// TIA Portal project "定时器练习，控制主轴电机和油泵电机的1顺序启停_V16" (V16)

(* hardware
DEVICE "S7-1200 station_1"  S7-1200 Station
   slot 0: "Rack_0"  S7-1200 Rack  Rack  V1.0
   slot 1: "PLC_1"  CPU 1214C DC/DC/DC  6ES7 214-1AG40-0XB0  V4.2
DEVICE "HMI_1"  KTP700 Basic PN
   slot 0: "HMI_1"  KTP700 Basic PN  6AV2 123-2GB03-0AX0  15.1.0.0
   slot 1: "HMI_RT_1"  KTP700 Basic PN  6AV2 123-2GB03-0AX0  15.1.0.0
   slot 5: "HMI_1.IE_CP_1"  PROFINET Interface  15.0.1.0
      slot 1: "PROFINET Interface_1"  PROFINET Interface
         slot 1: "Port_1"  Port
*)

// ===== PLC "PLC_1"  CPU 1214C DC/DC/DC =====

VAR_GLOBAL   // PLC tag table "默认变量表"
   "启动上升沿信号" AT %M0.0 : Bool;
   "油泵启动标志" AT %M0.1 : Bool;
   "启动电机延时信号" AT %MD200 : Time;
   "主轴标志" AT %M0.2 : Bool;
   "急停下降沿信号" AT %M0.3 : Bool;
   "油泵停止标志" AT %M0.4 : Bool;
   "主轴停止延时" AT %MD2004 : Time;
   "油泵停止标志(1)" AT %M0.5 : Bool;
   "上一个扫描周期" AT %M10.0 : Bool;
   "主轴标志1" AT %M10.1 : Bool;
   "油泵停止扫描周期" AT %M0.6 : Bool;
   "Tag_1" AT %M20.0 : Bool;
   "Tag_2" AT %M20.1 : Bool;
   "Tag_3" AT %M20.2 : Bool;
   "Tag_4" AT %M30.0 : Bool;
   "Tag_5" AT %M30.1 : Bool;
   "Tag_6" AT %M20.4 : Bool;
   "Tag_7" AT %M20.3 : Bool;
   "系统运行指示灯标志1" AT %M40.0 : Bool;
   "系统运行指示灯标志2" AT %M40.1 : Bool;
   "Tag_8" AT %MD300 : Time;
   "Tag_9" AT %MD304 : Time;
   "Tag_10" AT %MD308 : Time;
   "Tag_11" AT %MD312 : Time;
   "系统停止运行标志1" AT %M40.2 : Bool;
END_VAR

VAR_GLOBAL   // PLC tag table "io表"
   "启动" AT %I0.0 : Bool;
   "停止" AT %I0.1 : Bool;
   "正转" AT %I0.2 : Bool;
   "反转" AT %I0.3 : Bool;
   "急停" AT %I0.4 : Bool;
   "主轴急停" AT %I0.5 : Bool;
   "油泵电机急停" AT %I0.6 : Bool;
   "主轴继电器" AT %Q0.0 : Bool;
   "油泵继电器" AT %Q0.1 : Bool;
   "主轴正转" AT %Q0.2 : Bool;
   "主轴反转" AT %Q0.3 : Bool;
   "系统运行指示灯" AT %Q0.4 : Bool;
   "系统停止指示灯" AT %Q0.5 : Bool;
   "主轴运行指示灯" AT %Q0.6 : Bool;
   "油泵运行指示灯" AT %Q0.7 : Bool;
END_VAR

VAR_GLOBAL   // PLC tag table "触摸屏变量"
   "触摸屏启动" AT %M100.0 : Bool;
   "触摸屏停止" AT %M100.1 : Bool;
   "触摸屏急停" AT %M100.2 : Bool;
   "触摸屏正转" AT %M100.3 : Bool;
   "触摸屏反转" AT %M100.4 : Bool;
   "触摸屏正转急停" AT %M100.5 : Bool;
   "触摸屏反转急停" AT %M100.6 : Bool;
END_VAR

// folder: System blocks/Program resources

DATA_BLOCK "IEC_Timer_0_DB"   // DB1
{ S7_Optimized_Access := 'TRUE' }
AUTHOR : Simatic
FAMILY : IEC
NAME : IEC_TMR
VERSION : 1.0
// stored: InstanceOfName IEC_TIMER
"IEC_TIMER"
BEGIN
END_DATA_BLOCK

DATA_BLOCK "IEC_Timer_0_DB_1"   // DB2
{ S7_Optimized_Access := 'TRUE' }
AUTHOR : Simatic
FAMILY : IEC
NAME : IEC_TMR
VERSION : 1.0
// stored: InstanceOfName IEC_TIMER
"IEC_TIMER"
BEGIN
END_DATA_BLOCK

DATA_BLOCK "IEC_Timer_0_DB_2"   // DB3
{ S7_Optimized_Access := 'TRUE' }
AUTHOR : Simatic
FAMILY : IEC
NAME : IEC_TMR
VERSION : 1.0
// stored: InstanceOfName IEC_TIMER
"IEC_TIMER"
BEGIN
END_DATA_BLOCK

DATA_BLOCK "IEC_Timer_0_DB_3"   // DB4
{ S7_Optimized_Access := 'TRUE' }
AUTHOR : Simatic
FAMILY : IEC
NAME : IEC_TMR
VERSION : 1.0
// stored: InstanceOfName IEC_TIMER
"IEC_TIMER"
BEGIN
END_DATA_BLOCK

DATA_BLOCK "IEC_Timer_0_DB_4"   // DB5
{ S7_Optimized_Access := 'TRUE' }
AUTHOR : Simatic
FAMILY : IEC
NAME : IEC_TMR
VERSION : 1.0
// stored: InstanceOfName IEC_TIMER
"IEC_TIMER"
BEGIN
END_DATA_BLOCK

DATA_BLOCK "IEC_Timer_0_DB_5"   // DB6
{ S7_Optimized_Access := 'TRUE' }
AUTHOR : Simatic
FAMILY : IEC
NAME : IEC_TMR
VERSION : 1.0
// stored: InstanceOfName IEC_TIMER
"IEC_TIMER"
BEGIN
END_DATA_BLOCK

// folder: (top level)

ORGANIZATION_BLOCK "Main"   // OB1, LAD, ProgramCycle
TITLE = "Main Program Sweep (Cycle)"
{ S7_Optimized_Access := 'TRUE' }
VERSION : 0.1
   VAR_INPUT
      Initial_Call : Bool;   // Initial call of this OB
      Remanence : Bool;   // =True, if remanent data are available
   END_VAR
   VAR_TEMP   // added for the SCL form of the ladder/FBD networks
      _w1 : Bool;
      _w2 : Bool;
      _w3 : Bool;
      _w4 : Bool;
   END_VAR
BEGIN

REGION Network 1: 启动系统
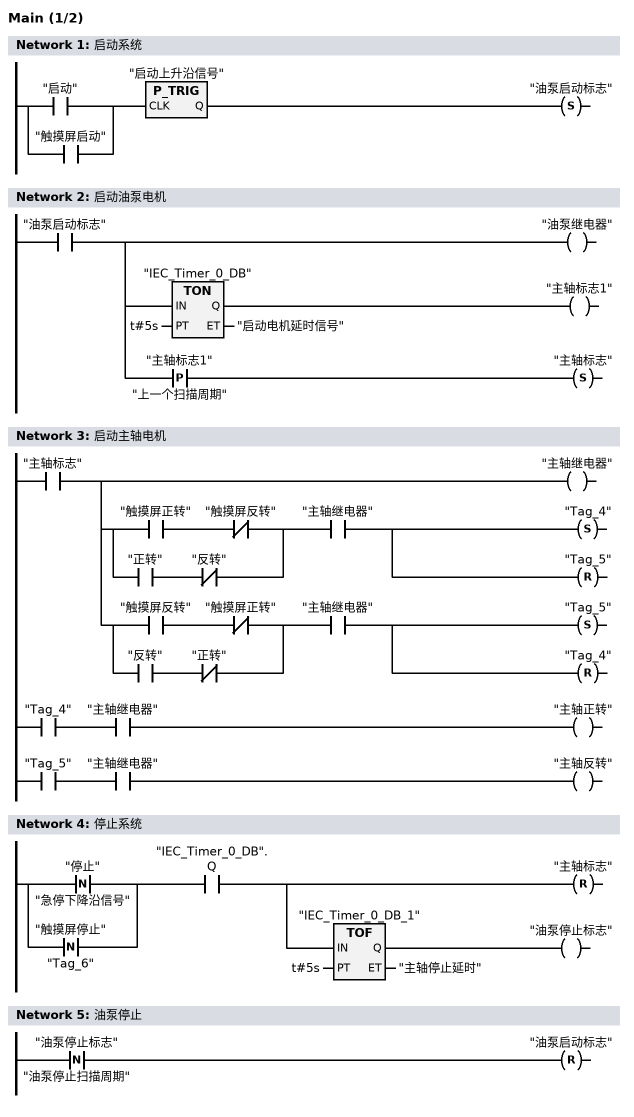
   RUNG wire#powerrail
      Contact( "启动" )
      wire#w1
      P_Trig( "启动上升沿信号" )
      S_Coil( "油泵启动标志" )
   END_RUNG
   RUNG wire#powerrail
      Contact( "触摸屏启动" )
   END_RUNG wire#w1
   // the same network as SCL:
   #_w1 := "启动" OR "触摸屏启动";
   #_w2 := #_w1 AND NOT "启动上升沿信号";   // rising edge
   "启动上升沿信号" := #_w1;
   IF #_w2 THEN "油泵启动标志" := TRUE; END_IF;
END_REGION

REGION Network 2: 启动油泵电机
   "油泵继电器" := "油泵启动标志";
   "IEC_Timer_0_DB".TON(IN := "油泵启动标志", PT := t#5s, ET => "启动电机延时信号");
   "主轴标志1" := "IEC_Timer_0_DB".Q;
   #_w1 := "油泵启动标志" AND "主轴标志1" AND NOT "上一个扫描周期";   // rising edge of "主轴标志1"
   "上一个扫描周期" := "主轴标志1";
   IF #_w1 THEN "主轴标志" := TRUE; END_IF;
END_REGION

REGION Network 3: 启动主轴电机
   RUNG wire#powerrail
      Contact( "主轴标志" )
      wire#w1
      Coil( "主轴继电器" )
   END_RUNG
   RUNG wire#w1
      Contact( "触摸屏正转" )
      I_Contact( "触摸屏反转" )
      wire#w2
      Contact( "主轴继电器" )
      wire#w3
      S_Coil( "Tag_4" )
   END_RUNG
   RUNG wire#w1
      Contact( "正转" )
      I_Contact( "反转" )
   END_RUNG wire#w2
   RUNG wire#w3
      R_Coil( "Tag_5" )
   END_RUNG
   RUNG wire#w1
      Contact( "触摸屏反转" )
      I_Contact( "触摸屏正转" )
      wire#w4
      Contact( "主轴继电器" )
      wire#w5
      S_Coil( "Tag_5" )
   END_RUNG
   RUNG wire#w1
      Contact( "反转" )
      I_Contact( "正转" )
   END_RUNG wire#w4
   RUNG wire#w5
      R_Coil( "Tag_4" )
   END_RUNG
   RUNG wire#powerrail
      Contact( "Tag_4" )
      Contact( "主轴继电器" )
      Coil( "主轴正转" )
   END_RUNG
   RUNG wire#powerrail
      Contact( "Tag_5" )
      Contact( "主轴继电器" )
      Coil( "主轴反转" )
   END_RUNG
   // the same network as SCL:
   "主轴继电器" := "主轴标志";
   IF "主轴标志" AND (("触摸屏正转" AND NOT "触摸屏反转") OR ("正转" AND NOT "反转")) AND "主轴继电器" THEN
       "Tag_4" := TRUE;
       "Tag_5" := FALSE;
   END_IF;
   IF "主轴标志" AND (("触摸屏反转" AND NOT "触摸屏正转") OR ("反转" AND NOT "正转")) AND "主轴继电器" THEN
       "Tag_5" := TRUE;
       "Tag_4" := FALSE;
   END_IF;
   "主轴正转" := "Tag_4" AND "主轴继电器";
   "主轴反转" := "Tag_5" AND "主轴继电器";
END_REGION

REGION Network 4: 停止系统
   #_w1 := NOT "停止" AND "急停下降沿信号";   // falling edge of "停止"
   "急停下降沿信号" := "停止";
   #_w2 := NOT "触摸屏停止" AND "Tag_6";   // falling edge of "触摸屏停止"
   "Tag_6" := "触摸屏停止";
   #_w3 := (#_w1 OR #_w2) AND "IEC_Timer_0_DB".Q;
   IF #_w3 THEN "主轴标志" := FALSE; END_IF;
   "IEC_Timer_0_DB_1".TOF(IN := #_w3, PT := t#5s, ET => "主轴停止延时");
   "油泵停止标志" := "IEC_Timer_0_DB_1".Q;
END_REGION

REGION Network 5: 油泵停止
   RUNG wire#powerrail
      N_Contact(operand := "油泵停止标志", bit := "油泵停止扫描周期")
      R_Coil( "油泵启动标志" )
   END_RUNG
   // the same network as SCL:
   #_w1 := NOT "油泵停止标志" AND "油泵停止扫描周期";   // falling edge of "油泵停止标志"
   "油泵停止扫描周期" := "油泵停止标志";
   IF #_w1 THEN "油泵启动标志" := FALSE; END_IF;
END_REGION

REGION Network 6: 急停
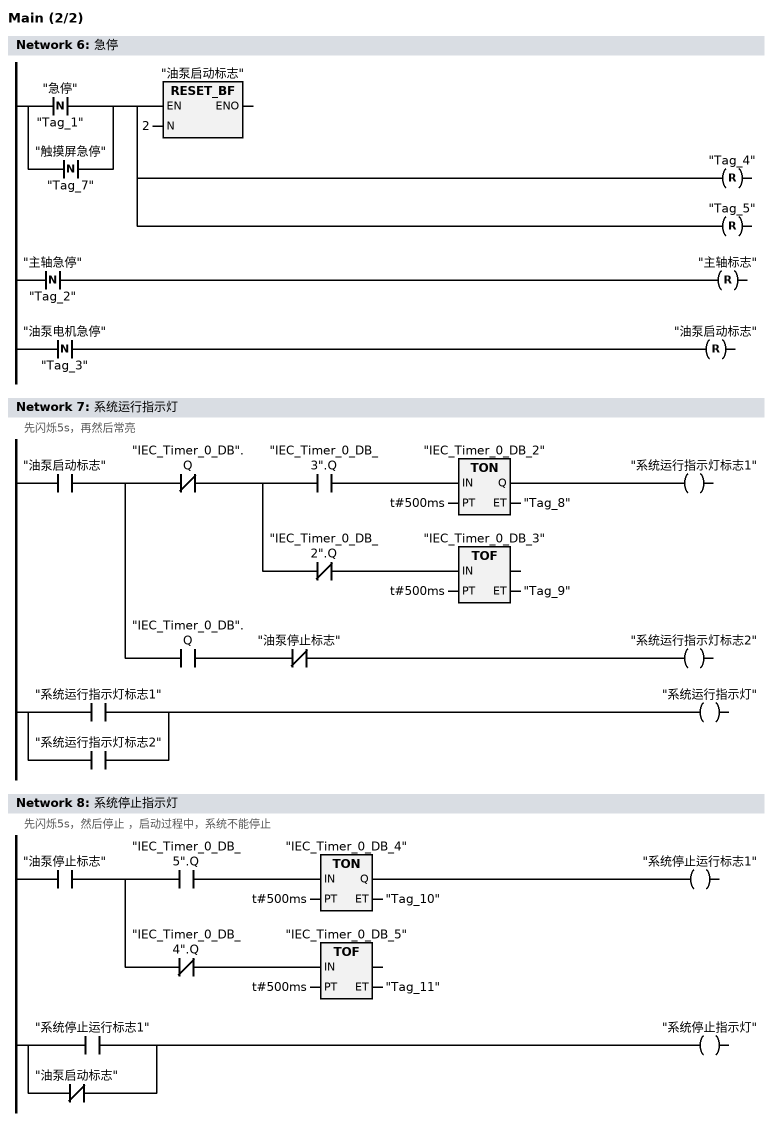
   // no SCL statement known for RBitfield: written as a call
   #_w1 := NOT "急停" AND "Tag_1";   // falling edge of "急停"
   "Tag_1" := "急停";
   #_w2 := NOT "触摸屏急停" AND "Tag_7";   // falling edge of "触摸屏急停"
   "Tag_7" := "触摸屏急停";
   IF #_w1 OR #_w2 THEN
       RESET_BF(operand := "油泵启动标志", n := 2);
       "Tag_4" := FALSE;
       "Tag_5" := FALSE;
   END_IF;
   #_w3 := NOT "主轴急停" AND "Tag_2";   // falling edge of "主轴急停"
   "Tag_2" := "主轴急停";
   IF #_w3 THEN "主轴标志" := FALSE; END_IF;
   #_w4 := NOT "油泵电机急停" AND "Tag_3";   // falling edge of "油泵电机急停"
   "Tag_3" := "油泵电机急停";
   IF #_w4 THEN "油泵启动标志" := FALSE; END_IF;
END_REGION

REGION Network 7: 系统运行指示灯
   // 先闪烁5s，再然后常亮
   #_w1 := "油泵启动标志" AND NOT "IEC_Timer_0_DB".Q;
   "IEC_Timer_0_DB_2".TON(IN := #_w1 AND "IEC_Timer_0_DB_3".Q, PT := t#500ms, ET => "Tag_8");
   "系统运行指示灯标志1" := "IEC_Timer_0_DB_2".Q;
   "IEC_Timer_0_DB_3".TOF(IN := #_w1 AND NOT "IEC_Timer_0_DB_2".Q, PT := t#500ms, ET => "Tag_9");
   "系统运行指示灯标志2" := "油泵启动标志" AND "IEC_Timer_0_DB".Q AND NOT "油泵停止标志";
   "系统运行指示灯" := "系统运行指示灯标志1" OR "系统运行指示灯标志2";
END_REGION

REGION Network 8: 系统停止指示灯
   // 先闪烁5s，然后停止 ，启动过程中，系统不能停止
   "IEC_Timer_0_DB_4".TON(IN := "油泵停止标志" AND "IEC_Timer_0_DB_5".Q, PT := t#500ms, ET => "Tag_10");
   "系统停止运行标志1" := "IEC_Timer_0_DB_4".Q;
   "IEC_Timer_0_DB_5".TOF(IN := "油泵停止标志" AND NOT "IEC_Timer_0_DB_4".Q, PT := t#500ms, ET => "Tag_11");
   "系统停止指示灯" := "系统停止运行标志1" OR NOT "油泵启动标志";
END_REGION
END_ORGANIZATION_BLOCK

(* ===== HMI "HMI_RT_1" =====
system functions are stored by id; their names below are inferred from use
connection "HMI_连接_1": ETHERNET, SMART_S7_1200_OMS

HMI tags "默认变量表"
   "Tag_ScreenNumber" : UInt, internal
   "触摸屏启动" : Bool = PLC 触摸屏启动 AT %M100.0, 100 ms
   "触摸屏停止" : Bool = PLC 触摸屏停止 AT %M100.1, 100 ms
   "触摸屏急停" : Bool = PLC 触摸屏急停 AT %M100.2, 100 ms
   "油泵继电器" : Bool = PLC 油泵继电器 AT %Q0.1, 100 ms
   "主轴继电器" : Bool = PLC 主轴继电器 AT %Q0.0, 100 ms
   "主轴正转" : Bool = PLC 主轴正转 AT %Q0.2, 100 ms
   "主轴反转" : Bool = PLC 主轴反转 AT %Q0.3, 100 ms
   "触摸屏正转" : Bool = PLC 触摸屏正转 AT %M100.3, 100 ms
   "触摸屏反转" : Bool = PLC 触摸屏反转 AT %M100.4, 100 ms
   "系统运行指示灯" : Bool = PLC 系统运行指示灯 AT %Q0.4, 100 ms
   "系统停止指示灯" : Bool = PLC 系统停止指示灯 AT %Q0.5, 100 ms

Template "模板_1" 800x480
   Button "退出" at 714,429 size 71x50; TextOff '退出'; PictureOff "ExitRuntime_KTP700_Basic_PN_TR"; PictureOn "ExitRuntime_KTP700_Basic_PN_TR"
      on Release: StopRuntime(0)
   Button "Template_Button" at 614,429 size 71x50; TextOff 'Text'
   Button "Template_Button_1" at 514,429 size 71x50; TextOff 'Text'
   Button "Template_Button_2" at 414,429 size 71x50; TextOff 'Text'
   Button "Template_Button_3" at 314,429 size 71x50; TextOff 'Text'
   Button "Template_Button_4" at 214,429 size 71x50; TextOff 'Text'
   Button "Template_Button_5" at 114,429 size 71x50; TextOff 'Text'
   Button "起始画面" at 14,429 size 71x50; TextOff '起始画面'; PictureOff "NavigateHome_KTP700_Basic_PN_TR"; PictureOn "NavigateHome_KTP700_Basic_PN_TR"
      on Release: ActivateScreen("根画面", 0)
   SymbolicIOField "Symbolic_IO_Field_Screen" at 93,9 size 600x33; TextOff '0'; TextOn '1'; TextList "TextList_ScreenNames"
      ProcessValue <- "Tag_ScreenNumber"
      on Change: ActivateScreenByNumber("Tag_ScreenNumber", 0)
   DateTimeField "HmiScreenItemData" at 695,25 size 105x25
   DateTimeField "HmiScreenItemData_1" at 695,0 size 105x25
   GraphicView "Logo" at 0,0 size 91x51; Picture "HMI_1 的 Logo"

screen "根画面" 800x480, template "模板_1"
   on GenerateScreen: SetTag("Tag_ScreenNumber", 1)
   TextField "HmiScreenItemData" at 98,223 size 640x25; Text 'Text'
   TextField "文本域_1" at 170,59 size 455x33; Text '主轴电机，油泵电机顺序启停控制'
   Button "按钮_1" at 25,121 size 96x32; TextOff '启动'
      on Press: SetBit("触摸屏启动")
      on Release: ResetBit("触摸屏启动")
   Button "按钮_2" at 23,195 size 96x32; TextOff '停止'
      on Press: SetBit("触摸屏停止")
      on Release: ResetBit("触摸屏停止")
   Button "按钮_3" at 23,296 size 96x32; TextOff '急停'
      on Press: SetBit("触摸屏急停")
      on Release: ResetBit("触摸屏急停")
   Button "按钮_4" at 660,305 size 96x32; TextOff '正转'
      on Press: SetBit("触摸屏正转")
      on Release: ResetBit("触摸屏正转")
   Button "按钮_5" at 655,378 size 96x32; TextOff '反转'
      on Press: SetBit("触摸屏反转")
      on Release: ResetBit("触摸屏反转")
   Circle "圆_1" at 279,161 size 48x48
      Appearance <- "油泵继电器"
   Circle "圆_2" at 376,163 size 48x48
      Appearance <- "主轴继电器"
   Circle "圆_3" at 665,121 size 48x48
      Appearance <- "主轴正转"
   Circle "圆_4" at 669,203 size 48x48
      Appearance <- "主轴反转"
   TextField "文本域_2" at 254,248 size 73x20; Text '油泵电机'
   TextField "文本域_3" at 363,245 size 73x20; Text '主轴电机'
   TextField "文本域_4" at 669,178 size 39x20; Text '正转'
   TextField "文本域_5" at 670,265 size 39x20; Text '反转'
   Circle "圆_5" at 65,349 size 24x24
      Appearance <- "系统运行指示灯"
   Circle "圆_6" at 65,393 size 25x25
      Appearance <- "系统停止指示灯"
   TextField "文本域_6" at 114,364 size 124x20; Text '系统运行指示灯'
*)